(*			
	RafalOS
	Rafał Osajda		22.12.2025		TC 4024.66
	Interejs łączacy kilka 
*)
INTERFACE ITF_Component2_HMI_Connector EXTENDS 
	ITF_BaseComponent_HMI_Connector, ITF_Component2_HMI_Connector_View, ITF_Component2_HMI_Connector_Command

END_INTERFACE

(* stored: Version 1.1.0.1
   Itf ITF_Component2_HMI_Connector: Id {fe7009d7-f5d1-026a-2b57-3890c9d2f854} *)
